FUNCTION_BLOCK FB_HMI_CALIBRATION_BEAM_SPLITTER EXTENDS FB_HMI_COMPONENT
VAR_INPUT
END_VAR
VAR_OUTPUT
END_VAR
VAR
END_VAR
VAR_IN_OUT
	{attribute 'OPC.UA.DA' := '0'}
	fbInstance		: FB_NOTT_CALIBRATION_BEAM_SPLITTER;


END_VAR


fbHealthStatus( 
				bIsEnabled:= TRUE, 
				bIsGood := NOT fbInstance.stat.bError,
				bHasWarning := fbInstance.stat.bWarning
				);
				
fbBusyStatus(
				bIsBusy := fbInstance.stat.bBusy,
				bIsEnabled := TRUE);
				
M_UpdateStatusColor();

END_FUNCTION_BLOCK

(* stored: Version 1.1.0.1, ProductVersion 3.1.4024.14
   POU FB_HMI_CALIBRATION_BEAM_SPLITTER: Id {509b4605-d229-44ee-ba8a-800c65136f56}, SpecialFunc None *)
